// TwinCAT 3 PLC project Untitled1
// ProgramVersion: 3.1.4026.16
// CompilerDefines: VISU_USEPROPERTYINFO
// libraries:
//   Tc2_Standard, * (Beckhoff Automation GmbH)
//   Tc2_System, * (Beckhoff Automation GmbH)
// project tree:
//   / GlobalTextList.TcGTLO, PlcTask.TcTTO, Visualization Manager.TcVMO (not stored)
//   POUs/ MAIN.TcPOU, MAIN_STL.TcPOU
//   VISUs/ Visualization.TcVIS
// real-time tasks:
//   TASK PlcTask: cycle T#10ms, priority 20, ADS port 350

CONFIGURATION Untitled1
    RESOURCE PLC ON TwinCAT3
        TASK PlcTask(INTERVAL := T#10ms, PRIORITY := 20);
        PROGRAM MAIN WITH PlcTask : MAIN;
    END_RESOURCE
END_CONFIGURATION

// ---- POUs/MAIN.TcPOU
PROGRAM MAIN
VAR_INPUT
	// Nostimen tulot
	iElevatorSensor AT %IX1.0: BOOL; // nostimen valoanturi
	iElevatorIsLifted AT %IX1.1: BOOL; // nostin on ajettu ylärajalle
	iElevatorIsDescended AT %IX1.2: BOOL; // nostin on ajettu alarajalle
	iElevatorConveyorRunning AT %IX1.3: BOOL; // nostimen kuljetin pyörii
	
	// Kuljetin 2 tulot
	iConveyor2Sensor AT %IX2.0: BOOL; // Valokenno kuljetin 2 ennen työnnintä
	iPusherPushed AT %IX2.1: BOOL; // Työnnnin on ulkona
	iPusherRetracted AT %IX2.2: BOOL; // Työnnin on sisällä
	iConveyor2Running AT %IX2.3: BOOL; // kuljetin 2 pyörii
	
	// Kuljetin 1 tulot
	iConveyor1Running AT %IX3.0: BOOL; // Kuljetin 1 pyörii
END_VAR

VAR_OUTPUT
	// Kuljetin 1 lähdöt
	qConveyor1 AT %QX0.0: BOOL; // Kuljetin 1 ajo
	
	// Nostimen lähdöt
	qElevatorConveyor AT %QX1.0: BOOL; // Nostimen kuljetin ajo
	qElevatorUp AT %QX1.1: BOOL; // Nostimen nosto ylös
	qElevatorDown AT %QX1.2: BOOL; // Nostimen lasku alas
	
	// Kuljetin 2 lähdöt
	qConveyor2 AT %QX2.0: BOOL; // Kuljetin 2 ajo 
	qPusherPush AT %QX2.1: BOOL; // Työnnin eteen
	qPusherRetract AT %QX2.2: BOOL; // Työnnin taakse
	
	// Laatikon lähtö 
	qBoxShaker AT %QX3.0: BOOL; // Laatikon tärytin
END_VAR

VAR
	ManConveyor1: BOOL; // Kuljetin 1 ajo
	ManElevatorConveyor: BOOL; // Nostimen kuljetin ajo
	ManElevatorUp: BOOL; // Nostimen nosto ylös
	ManElevatorDown: BOOL; // Nostimen lasku alas
	ManConveyor2: BOOL; // Kuljetin 2 ajo 
	ManPusherPush: BOOL; // Työnnin eteen
	ManPusherRetract: BOOL; // Työnnin taakse
	ManBoxShaker: BOOL; // Laatikon tärytin	
	Manual_mode: BOOL;
	Auto_mode: BOOL;
	Lamp: BOOL;
	START: BOOL;
	Seq1: BOOL;
	Seq2: BOOL;
	Seq3: BOOL;
	Seq4: BOOL;
	Seq5: BOOL;
	STOP: BOOL;
END_VAR
VAR // added by the converter: edge detectors and wires of the graphical bodies
    _ft1 : F_TRIG;
    _w1 : BOOL;
END_VAR

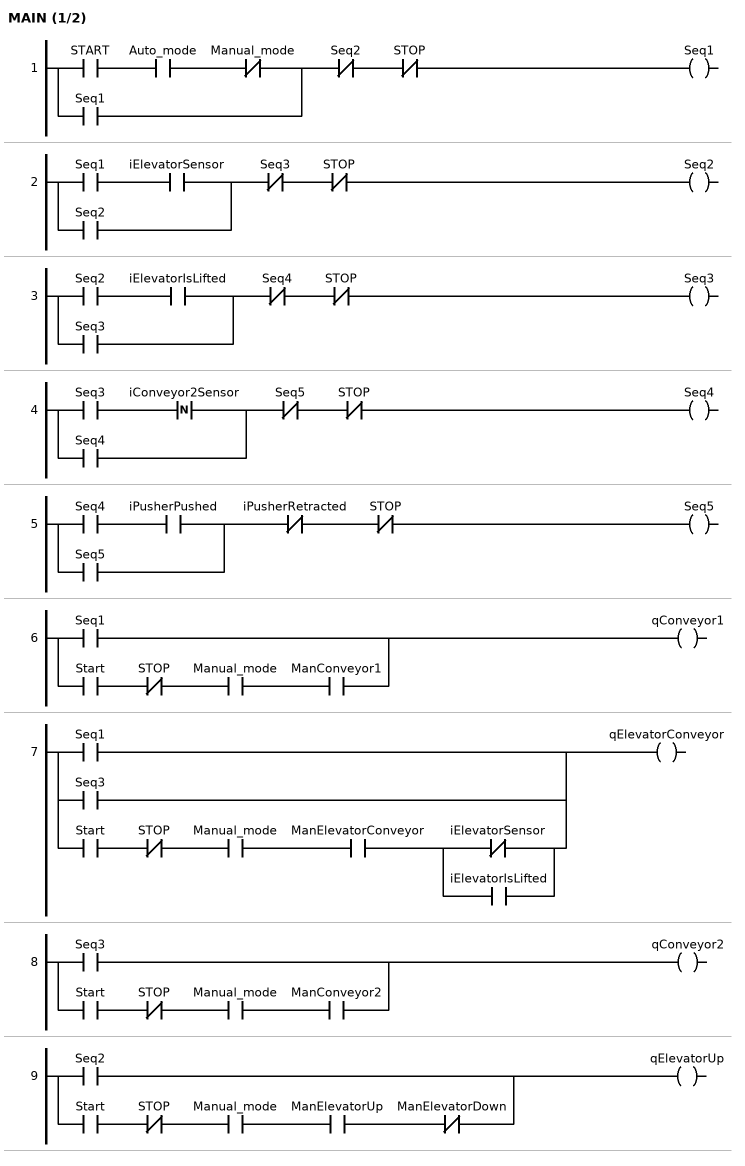
// NETWORK 1
Seq1 := (START AND Auto_mode AND NOT Manual_mode OR Seq1) AND NOT Seq2 AND NOT STOP;

// NETWORK 2
Seq2 := (Seq1 AND iElevatorSensor OR Seq2) AND NOT Seq3 AND NOT STOP;

// NETWORK 3
Seq3 := (Seq2 AND iElevatorIsLifted OR Seq3) AND NOT Seq4 AND NOT STOP;

// NETWORK 4
_ft1(CLK := iConveyor2Sensor);
Seq4 := (Seq3 AND _ft1.Q OR Seq4) AND NOT Seq5 AND NOT STOP;

// NETWORK 5
Seq5 := (Seq4 AND iPusherPushed OR Seq5) AND NOT iPusherRetracted AND NOT STOP;

// NETWORK 6
qConveyor1 := Seq1 OR Start AND NOT STOP AND Manual_mode AND ManConveyor1;

// NETWORK 7
_w1 := Start AND NOT STOP AND Manual_mode AND ManElevatorConveyor;
qElevatorConveyor := Seq1 OR Seq3 OR (_w1 AND NOT iElevatorSensor OR _w1 AND iElevatorIsLifted);

// NETWORK 8
qConveyor2 := Seq3 OR Start AND NOT STOP AND Manual_mode AND ManConveyor2;

// NETWORK 9
qElevatorUp := Seq2 OR Start AND NOT STOP AND Manual_mode AND ManElevatorUp AND NOT ManElevatorDown;

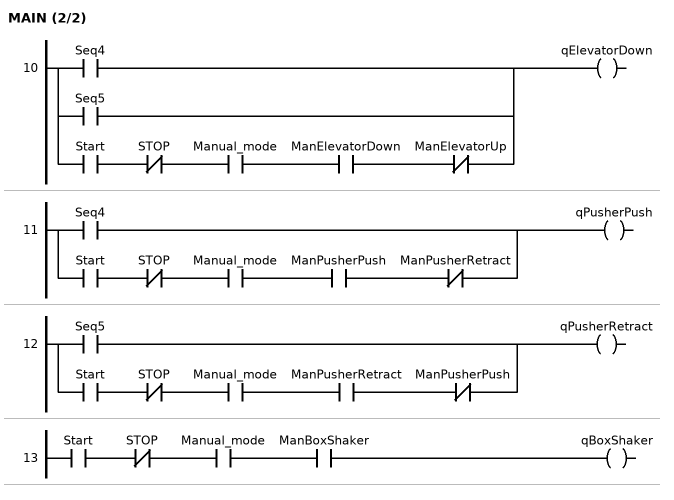
// NETWORK 10
qElevatorDown := Seq4 OR Seq5 OR Start AND NOT STOP AND Manual_mode AND ManElevatorDown AND NOT ManElevatorUp;

// NETWORK 11
qPusherPush := Seq4 OR Start AND NOT STOP AND Manual_mode AND ManPusherPush AND NOT ManPusherRetract;

// NETWORK 12
qPusherRetract := Seq5 OR Start AND NOT STOP AND Manual_mode AND ManPusherRetract AND NOT ManPusherPush;

// NETWORK 13
qBoxShaker := Start AND NOT STOP AND Manual_mode AND ManBoxShaker;

END_PROGRAM

// ---- POUs/MAIN_STL.TcPOU
PROGRAM MAIN_STL
VAR
		// Nostimen tulot
	iElevatorSensor AT %IX1.0: BOOL; // nostimen valoanturi
	iElevatorIsLifted AT %IX1.1: BOOL; // nostin on ajettu ylärajalle
	iElevatorIsDescended AT %IX1.2: BOOL; // nostin on ajettu alarajalle
	iElevatorConveyorRunning AT %IX1.3: BOOL; // nostimen kuljetin pyörii
	
	// Kuljetin 2 tulot
	iConveyor2Sensor AT %IX2.0: BOOL; // Valokenno kuljetin 2 ennen työnnintä
	iPusherPushed AT %IX2.1: BOOL; // Työnnnin on ulkona
	iPusherRetracted AT %IX2.2: BOOL; // Työnnin on sisällä
	iConveyor2Running AT %IX2.3: BOOL; // kuljetin 2 pyörii
	
	// Kuljetin 1 tulot
	iConveyor1Running AT %IX3.0: BOOL; // Kuljetin 1 pyörii
	
		// Kuljetin 1 lähdöt
	qConveyor1 AT %QX0.0: BOOL; // Kuljetin 1 ajo
	
	// Nostimen lähdöt
	qElevatorConveyor AT %QX1.0: BOOL; // Nostimen kuljetin ajo
	qElevatorUp AT %QX1.1: BOOL; // Nostimen nosto ylös
	qElevatorDown AT %QX1.2: BOOL; // Nostimen lasku alas
	
	// Kuljetin 2 lähdöt
	qConveyor2 AT %QX2.0: BOOL; // Kuljetin 2 ajo 
	qPusherPush AT %QX2.1: BOOL; // Työnnin eteen
	qPusherRetract AT %QX2.2: BOOL; // Työnnin taakse
	
	// Laatikon lähtö 
	qBoxShaker AT %QX3.0: BOOL; // Laatikon tärytin
END_VAR

END_PROGRAM

// ---- GlobalTextList.TcGTLO
TEXTLIST GlobalTextList
  969 = 'Auto'
  83 = 'Auto mode'
  731 = 'Auto_mode'
  703 = 'Box shaker'
  960 = 'Conv1'
  792 = 'Conv2'
  790 = 'Convey '
  812 = 'Conveyor 1 '
  21 = 'Conveyor 2'
  634 = 'Conveyor 2 sensor'
  128 = 'Conveyor Belt 1'
  764 = 'Conveyor Belt 2'
  645 = 'Conveyor Belt 3'
  68 = 'dfsfs'
  397 = 'down'
  578 = 'Elevator  '
  384 = 'Elevator Conveyor'
  415 = 'Elevator Down'
  852 = 'Elevator down'
  3 = 'Elevator sensor'
  980 = 'Elevator up'
  387 = 'Elevator Up '
  976 = 'ertertert'
  357 = 'For example: Disable the elevator up before clicking the elevator down and the same for push out and pull back'
  780 = 'Manual'
  426 = 'Manual mode'
  498 = 'Mode'
  179 = 'NOTICE: You will have to disable the button which has the opposite state before activating the other one.'
  207 = 'NOTICE: You will have to disable the button which has the opposite state before activating the other one.\n'
  977 = 'Pull back'
  642 = 'push'
  113 = 'Push out'
  163 = 'Pusher push'
  963 = 'Pusher retract'
  622 = 'Reset'
  96 = 'retract'
  646 = 'Sensor 1'
  725 = 'Sensor 2'
  767 = 'START'
  63 = 'Start'
  20 = 'Stop'
  607 = 'Test lamp for the user interface'
  107 = 'up'
END_TEXTLIST

// ---- VISUs/Visualization.TcVIS
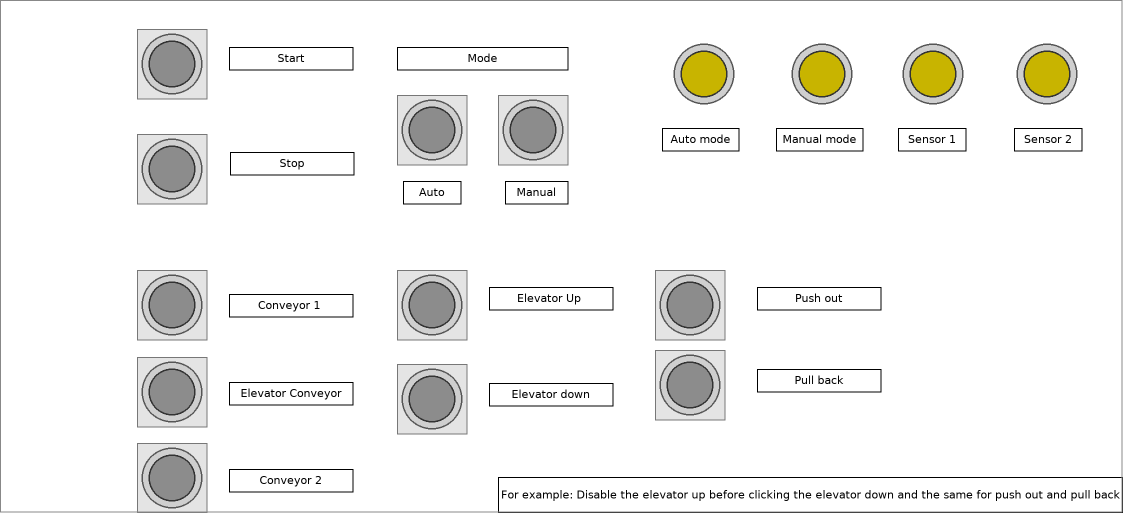
VISUALIZATION Visualization  // 1123x513
AR_IN_OUT
AR_IN_OUT
	
END_VAR
    PushSwitch (137,29 70x70), tooltip "START", variable: MAIN.START, behaviour: TOGGLE, style: Switch-PushSwitch-Gray
    PushSwitch (137,134 70x70), tooltip "Stop", variable: MAIN.STOP, behaviour: TOGGLE, style: Switch-PushSwitch-Gray
    PushSwitch (137,270 70x70), tooltip "Conv1", variable: MAIN.ManConveyor1, behaviour: TOGGLE, style: Switch-PushSwitch-Gray
    PushSwitch (137,443 70x70), tooltip "Conv2", variable: MAIN.ManConveyor2, behaviour: TOGGLE, style: Switch-PushSwitch-Gray
    PushSwitch (397,270 70x70), tooltip "up", variable: MAIN.ManElevatorUp, behaviour: TOGGLE, style: Switch-PushSwitch-Gray
    PushSwitch (397,364 70x70), tooltip "down", variable: MAIN.ManElevatorDown, behaviour: TOGGLE, style: Switch-PushSwitch-Gray
    PushSwitch (655,270 70x70), tooltip "push", variable: MAIN.ManPusherPush, behaviour: TOGGLE, style: Switch-PushSwitch-Gray
    PushSwitch (655,350 70x70), tooltip "retract", variable: MAIN.ManPusherRetract, behaviour: TOGGLE, style: Switch-PushSwitch-Gray
    PushSwitch (397,95 70x70), tooltip "Auto_mode", variable: MAIN.Auto_mode, behaviour: TOGGLE, style: Switch-PushSwitch-Gray
    PushSwitch (498,95 70x70), tooltip "Manual mode", variable: MAIN.Manual_mode, behaviour: TOGGLE, style: Switch-PushSwitch-Gray
    PushSwitch (137,357 70x70), tooltip "Conv1", variable: MAIN.ManElevatorConveyor, behaviour: TOGGLE, style: Switch-PushSwitch-Gray
    Rectangle (397,47 171x23), "Mode"
    Rectangle (403,181 58x23), "Auto"
    Rectangle (505,181 63x23), "Manual"
    Rectangle (229,47 124x23), "Start"
    Rectangle (230,152 124x23), "Stop"
    Rectangle (229,294 124x23), "Conveyor 1"
    Rectangle (229,382 124x23), "Elevator Conveyor"
    Rectangle (489,287 124x23), "Elevator Up"
    Rectangle (489,383 124x23), "Elevator down"
    Rectangle (229,469 124x23), "Conveyor 2"
    Rectangle (757,287 124x23), "Push out"
    Rectangle (757,369 124x23), "Pull back"
    Lamp1 (1012,39 70x70), variable: MAIN.iConveyor2Sensor, style: Lamp-Lamp1-Yellow
    Lamp1 (898,39 70x70), variable: MAIN.iElevatorSensor, style: Lamp-Lamp1-Yellow
    Rectangle (898,128 68x23), "Sensor 1"
    Rectangle (1014,128 68x23), "Sensor 2"
    Lamp1 (669,39 70x70), variable: MAIN.Auto_mode, style: Lamp-Lamp1-Yellow
    Lamp1 (787,39 70x70), variable: MAIN.Manual_mode, style: Lamp-Lamp1-Yellow
    Rectangle (662,128 77x23), "Auto mode"
    Rectangle (776,128 87x23), "Manual mode"
    Rectangle (498,477 625x36), "For example: Disable the elevator up before clicking the elevator down and the same for push out and pull back"
END_VISUALIZATION
